Universal Robots PolyScope program: forcegroup2.urp

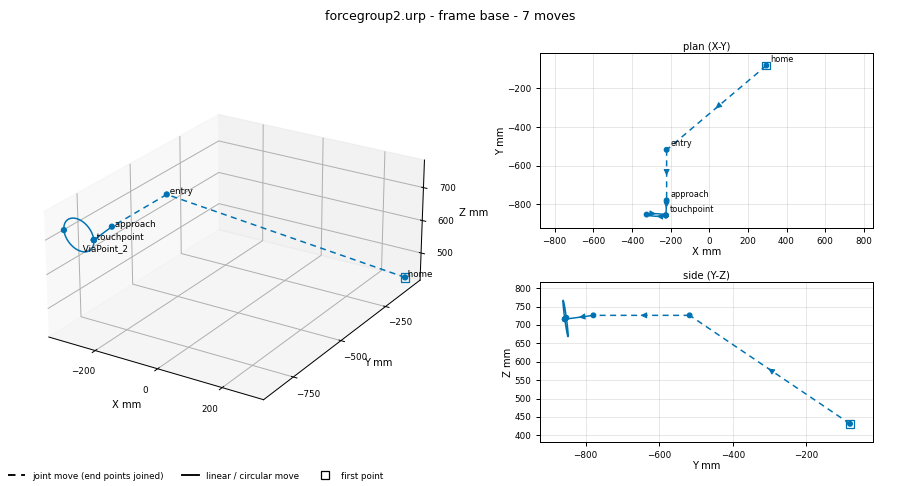
[picture p0: tool path of forcegroup2.urp in frame base, 7 of 9 moves have a stored position in this frame; points joined in program order, loops and branches not executed]
Program forcegroup2 (installation=group_2 directory=/programs/usbdisk_0 createdIn=5.12.4.1101661 lastSavedIn=5.12.4.1101661 robotSerialNumber=20205000194)
Calibrated DH parameters: a=[-0.000072, -0.302179, -0.53618, -0.000002, -0.000085, 0]; d=[0.181029, 536.296696, -453.808941, -82.313641, 0.119922, 0.115618]; alpha=[1.57037, -0.000994, -0.002401, 1.569923, -1.570986, 0]; deltaTheta=[0, -1.055132, 6.984537, 0.353782, -0.000001, 0]
Robot Program (runOnlyOnce=true)
  Folder pre_start
    Set NoAction tcp=marker_tip
    URCap Gripper (Robotiq_Grippers, Robotiq Inc.) dataModel(position=100.0, force=0.0, speed=0.0, positionInDouble=100.0, forceInDouble=0.0, speedInDouble=0.0, slaveIds=[9], blocking=true)
    MoveJ speed 60 deg/s, acceleration 80 deg/s^2 (useActiveTCP=true) feature=Base
      Waypoint home: motionParameters(nextMotionTime=2); TCP in base x=295.727 y=-81.103 z=431.152 mm, rx=-0.315 ry=3.1085 rz=0.0153 rad; joints [20.588, -45.93, -117.038, -105.93, 90.164, 99.013] deg; TCP offset x=-2.447 y=-7.658 z=243.941 mm, rx=0 ry=0 rz=0 rad
  Folder enter_wb
    MoveJ speed 60 deg/s, acceleration 80 deg/s^2 (useActiveTCP=true) feature=Base
      Waypoint entry: TCP in base x=-220.519 y=-517.31 z=726.121 mm, rx=0.963 ry=1.533 rz=-1.5405 rad; joints [-99.891, -62.475, -129.468, 12.005, 99.592, 63.789] deg; TCP offset x=0 y=0 z=160 mm, rx=0 ry=0 rz=0 rad
  Folder appr_wb
    MoveJ speed 60 deg/s, acceleration 80 deg/s^2 (useActiveTCP=true) feature=Base
      Waypoint approach: TCP in base x=-220.514 y=-778.948 z=726.137 mm, rx=1.2137 ry=1.2033 rz=-1.2118 rad; joints [-94.997, -88.213, -110.916, 19.206, 94.733, 90] deg; TCP offset x=0 y=0 z=160 mm, rx=0 ry=0 rz=0 rad
  Folder draw_on_wb
    MoveL speed 250 mm/s, acceleration 1200 mm/s^2 (useActiveTCP=true) feature=Base
      Waypoint touchpoint: TCP in base x=-224.155 y=-856.774 z=715.649 mm, rx=1.2137 ry=1.2033 rz=-1.2117 rad; joints [-94.691, -95.675, -104.281, 20.033, 94.438, 90] deg; TCP offset x=0 y=0 z=160 mm, rx=0 ry=0 rz=0 rad
    MoveP speed 250 mm/s, acceleration 1200 mm/s^2 (blendRadius=0.025 useActiveTCP=true) feature=Base
      Waypoint touchpoint: TCP in base x=-224.155 y=-856.774 z=715.649 mm, rx=1.2137 ry=1.2033 rz=-1.2117 rad; joints [-94.691, -95.675, -104.281, 20.033, 94.438, 90] deg
      CircleMove (OrientationMode=UNCONSTRAINED)
        Waypoint ViaPoint_1: TCP in base x=-272.536 y=-861.407 z=767.027 mm, rx=1.2137 ry=1.2033 rz=-1.2117 rad; joints [-99.151, -96.406, -98.066, 14.531, 98.888, 89.995] deg
        Waypoint EndPoint_1: TCP in base x=-323.995 y=-852.511 z=719.526 mm, rx=1.2136 ry=1.2032 rz=-1.2119 rad; joints [-103.904, -99.163, -99.874, 19.097, 103.651, 90.006] deg
      CircleMove (OrientationMode=UNCONSTRAINED)
        Waypoint ViaPoint_2: TCP in base x=-275.583 y=-847.89 z=668.232 mm, rx=1.2135 ry=1.2031 rz=-1.2118 rad; joints [-99.642, -98.564, -106.127, 24.769, 99.401, 90.014] deg
        Waypoint EndPoint_2: TCP in base x=-224.17 y=-856.727 z=715.78 mm, rx=1.2136 ry=1.2031 rz=-1.2118 rad; joints [-94.693, -95.67, -104.277, 20.033, 94.438, 90] deg
  SuppressedNode
    Folder return_to_start
      Placeholder
